FUNCTION_BLOCK MockObj IMPLEMENTS I_Cyclic, I_Initialise, I_Object, I_Resettable
VAR_INPUT
END_VAR
VAR_OUTPUT
END_VAR
VAR
END_VAR

METHOD Cycle : HRESULT
END_METHOD

METHOD Initialise : HRESULT
END_METHOD

METHOD RegisterWithParent
VAR_INPUT
	Runner	: I_HostObjects;
END_VAR
Runner.RegisterCyclic(THIS^);
Runner.RegisterInitialise(THIS^);
END_METHOD

METHOD Reset : Base_Library.HRESULT
END_METHOD

END_FUNCTION_BLOCK

(* stored: Version 1.1.0.1
   POU MockObj: Id {459c9319-db86-4d6a-b774-a97d62f0aee0}, SpecialFunc None
   Method Cycle: Id {2fdaa782-1cce-42d3-b0fd-0a553501ea73}
   Method Initialise: Id {b6fb438d-078a-4d9d-ba13-f31f733124cc}
   Method RegisterWithParent: Id {53309e55-7b39-4961-93ff-498d9c30e110}
   Method Reset: Id {fdee9a2d-cec1-4e56-8d77-d56933a1dff5} *)
